// TIA Portal V16 export
// export: Created 2021-08-30T13:41:02.1375407Z, ExportSetting WithDefaults, DisplayName Totally Integrated Automation Portal, DisplayVersion V16 Update 3, DisplayName TIA Portal Version Control Interface, DisplayVersion V16 Update 2, DisplayName TIA Portal Openness, DisplayVersion V16 Update 3, DisplayName TIA Portal Teamcenter Gateway, DisplayVersion V16, DisplayName STEP 7 Professional, DisplayVersion V16 Update 3, DisplayName STEP 7 Safety, DisplayVersion V16, DisplayName WinCC Advanced, DisplayVersion V16 Update 3
TYPE "DPump"
// stored: IsFailsafeCompliant false
   STRUCT
      mode : Bool;   // 1-ручной, 0-авто
      cmAuto { ExternalAccessible := 'False'; ExternalVisible := 'False'; ExternalWritable := 'False'} : Bool;   // авто команда
      cmHand : Bool;   // ручная команда
      block { ExternalAccessible := 'False'; ExternalVisible := 'False'; ExternalWritable := 'False'} : Bool;   // Внешняя блокировка
      service : Bool;   // Сервисный режим
      error { ExternalAccessible := 'False'; ExternalVisible := 'False'; ExternalWritable := 'False'} : Bool;   // Наличие любой ошибки
      showButton : Bool;   // 0- Показать, 1 - Скрыть
      feedBack { S7_SetPoint := 'True'} : Bool;   // Обратная связь
      st : Word;   // Состояние
      startTime { S7_SetPoint := 'True'} : Int := 5;   // Время запуска, сек
      stopTime { S7_SetPoint := 'True'} : Int := 5;   // Время останова, сек
      outCmStart { ExternalAccessible := 'False'; ExternalVisible := 'False'; ExternalWritable := 'False'} : Bool;   // Программный выход запуска насоса
      ack { ExternalAccessible := 'False'; ExternalVisible := 'False'; ExternalWritable := 'False'} : Word;   // Резерв
      spare1 : Word;
   END_STRUCT;
END_TYPE
